// TIA Portal V20 export
FUNCTION "SCurveProfile_Vision_Cal" : Void   // FC101, SCL
// stored: Access Published, SetENOAutomatically false
   VAR_INPUT
      CPM : LReal;
      travelDistance : LReal;
   END_VAR
   VAR_OUTPUT
      velocity : LReal;
      acceleration : LReal;
      deceleration : LReal;
      jerk : LReal;
   END_VAR
   VAR_TEMP
      CycleTime : LReal;
   END_VAR
   VAR CONSTANT
      PI : LReal := 3.14159265;
   END_VAR
BEGIN
   REGION Velocity
       #CycleTime := ((60.0 / #CPM) / 2.0) / 3.0;
       //#distance := #travelDistance;
       #velocity := 2.0 * #travelDistance / #CycleTime;
       #acceleration := #velocity * #PI / #CycleTime;
       #deceleration := #acceleration;
       #jerk := #velocity * 2 * #PI * #PI / (#CycleTime * #CycleTime);
   END_REGION
END_FUNCTION
